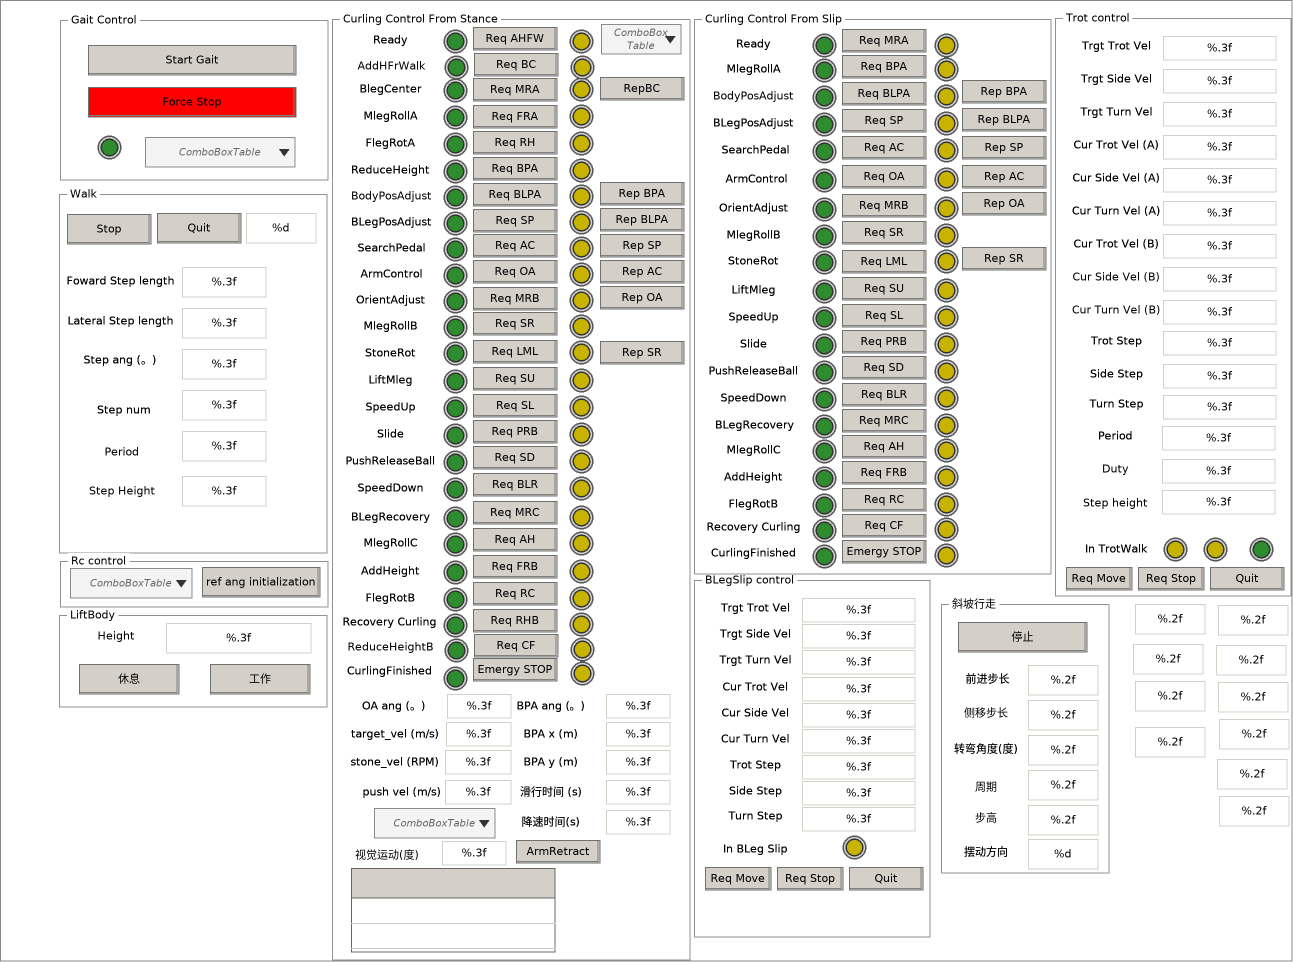
VISUALIZATION RobotUI  // 1293x962
    GroupBox (60,12 268x168), "Gait Control"
        Button (28,33 208x30), "Start Gait", input disabled if: GVL.isInGaitMode
            toggle GVL.startGaitButton
        Button (28,75 208x30), "Force Stop"
            toggle GVL.emergencyStop
        Lamp1 (36,121 27x29), variable: GVL.isInGaitMode, style: Lamp-Lamp1-Green
        ComboBoxTable (85,125 150x30), variable: GVL.gaitId, data array: GVL.gaitNameLists
            p3854506369: GVL.gaitNameLists[INDEX]
    Button (88,45 208x30), "Start Gait", input disabled if: GVL.isInGaitMode
        toggle GVL.startGaitButton
    Button (88,87 208x30), "Force Stop"
        toggle GVL.emergencyStop
    Lamp1 (96,133 27x29), variable: GVL.isInGaitMode, style: Lamp-Lamp1-Green
    ComboBoxTable (145,137 150x30), variable: GVL.gaitId, data array: GVL.gaitNameLists
        p3854506369: GVL.gaitNameLists[INDEX]
    GroupBox (59,186 268x367), "Walk"
        Button (8,28 84x30), "Stop"
            toggle GVL.gaitPlanner.StaticwalkGaitPlanner.require_stop_flag
        Button (98,27 84x30), "Quit"
            toggle GVL.gaitPlanner.StaticwalkGaitPlanner.quit_flag
        Textfield (123,81 84x30), "%.3f", text variable: GVL.gaitPlanner.StaticwalkGaitPlanner.L
            OnMouseClick: write the text variable via Default
        Label (8,80 107x30), "Foward Step length"
        Textfield (123,245 84x30), "%.3f", text variable: GVL.gaitPlanner.StaticwalkGaitPlanner.period
            OnMouseClick: write the text variable via Default
        Textfield (123,290 84x30), "%.3f", text variable: GVL.gaitPlanner.StaticwalkGaitPlanner.H
            OnMouseClick: write the text variable via Default
        Label (21,159 80x30), "Step ang (。)"
        Textfield (123,163 84x30), "%.3f", text variable: GVL.gaitPlanner.StaticwalkGaitPlanner.Yaw
            OnMouseClick: write the text variable via Default
        Label (25,209 80x30), "Step num"
        Textfield (123,204 84x30), "%.3f", text variable: GVL.gaitPlanner.StaticwalkGaitPlanner.N
            OnMouseClick: write the text variable via Default
        Textfield (123,122 84x30), "%.3f", text variable: GVL.gaitPlanner.StaticwalkGaitPlanner.La
            OnMouseClick: write the text variable via Default
        Label (8,120 107x30), "Lateral Step length"
    Button (67,214 84x30), "Stop"
        toggle GVL.gaitPlanner.StaticwalkGaitPlanner.require_stop_flag
    Button (157,213 84x30), "Quit"
        toggle GVL.gaitPlanner.StaticwalkGaitPlanner.quit_flag
    Textfield (182,267 84x30), "%.3f", text variable: GVL.gaitPlanner.StaticwalkGaitPlanner.L
        OnMouseClick: write the text variable via Default
    Label (67,266 107x30), "Foward Step length"
    Textfield (182,431 84x30), "%.3f", text variable: GVL.gaitPlanner.StaticwalkGaitPlanner.period
        OnMouseClick: write the text variable via Default
    Textfield (182,476 84x30), "%.3f", text variable: GVL.gaitPlanner.StaticwalkGaitPlanner.H
        OnMouseClick: write the text variable via Default
    Label (80,345 80x30), "Step ang (。)"
    Textfield (182,349 84x30), "%.3f", text variable: GVL.gaitPlanner.StaticwalkGaitPlanner.Yaw
        OnMouseClick: write the text variable via Default
    Label (84,395 80x30), "Step num"
    Textfield (182,390 84x30), "%.3f", text variable: GVL.gaitPlanner.StaticwalkGaitPlanner.N
        OnMouseClick: write the text variable via Default
    Textfield (182,308 84x30), "%.3f", text variable: GVL.gaitPlanner.StaticwalkGaitPlanner.La
        OnMouseClick: write the text variable via Default
    Label (67,306 107x30), "Lateral Step length"
    GroupBox (59,607 268x100), "LiftBody"
        Label (25,14 64x30), "Height"
        Textfield (107,16 145x30), "%.3f", text variable: GVL.ReduceDistance
            OnMouseClick: write the text variable via Default, min -0.3, max 0.3
        Button (20,57 100x30), "休息"
            toggle gvl.RestButton
        Button (151,57 100x30), "工作"
            toggle gvl.WorkButton
    Label (82,437 80x30), "Period"
    Label (77,476 90x30), "Step Height"
    Textfield (246,213 70x30), "%d", text variable: GVL.gaitPlanner.StaticwalkGaitPlanner.gait_cycle
    GroupBox (332,11 358x949), "Curling Control From Stance"
        Label (4,680 116x30), "OA ang (。)"
        Label (5,14 107x30), "Ready"
        Label (5,63 107x30), "BlegCenter"
        Label (5,90 107x30), "MlegRollA"
        Label (5,117 107x30), "FlegRotA"
        Label (5,144 107x30), "ReduceHeight"
        Label (5,300 107x30), "MlegRollB"
        Label (5,327 107x30), "StoneRot"
        Label (5,354 107x30), "LiftMleg"
        Label (5,381 107x30), "SpeedUp"
        Label (5,408 107x30), "Slide"
        Label (5,435 107x30), "PushReleaseBall"
        Label (5,462 107x30), "SpeedDown"
        Label (5,545 107x30), "AddHeight"
        Label (5,517 107x30), "MlegRollC"
        Label (5,572 107x30), "FlegRotB"
        Label (4,645 107x30), "CurlingFinished"
        Lamp1 (110,16 27x29), variable: GVL.gaitPlanner.CurlingGaitPlanner2.IsReady, style: Lamp-Lamp1-Green
        Lamp1 (110,65 27x29), variable: GVL.gaitPlanner.CurlingGaitPlanner2.IsBlegCenter, style: Lamp-Lamp1-Green
        Lamp1 (110,92 27x29), variable: GVL.gaitPlanner.CurlingGaitPlanner2.IsMlegRollA, style: Lamp-Lamp1-Green
        Lamp1 (110,119 27x29), variable: GVL.gaitPlanner.CurlingGaitPlanner2.IsFlegRotA, style: Lamp-Lamp1-Green
        Lamp1 (110,146 27x29), variable: GVL.gaitPlanner.CurlingGaitPlanner2.IsReduceHeight, style: Lamp-Lamp1-Green
        Lamp1 (110,302 27x29), variable: GVL.gaitPlanner.CurlingGaitPlanner2.IsMlegRollB, style: Lamp-Lamp1-Green
        Lamp1 (110,328 27x29), variable: GVL.gaitPlanner.CurlingGaitPlanner2.IsStoneRot, style: Lamp-Lamp1-Green
        Lamp1 (110,356 27x29), variable: GVL.gaitPlanner.CurlingGaitPlanner2.IsLiftMleg, style: Lamp-Lamp1-Green
        Lamp1 (110,383 27x29), variable: GVL.gaitPlanner.CurlingGaitPlanner2.IsSpeedUp, style: Lamp-Lamp1-Green
        Lamp1 (110,410 27x29), variable: GVL.gaitPlanner.CurlingGaitPlanner2.IsSlide, style: Lamp-Lamp1-Green
        Lamp1 (110,437 27x29), variable: GVL.gaitPlanner.CurlingGaitPlanner2.IsPushReleaseBall, style: Lamp-Lamp1-Green
        Lamp1 (110,464 27x29), variable: GVL.gaitPlanner.CurlingGaitPlanner2.IsSpeedDown, style: Lamp-Lamp1-Green
        Lamp1 (110,519 27x29), variable: GVL.gaitPlanner.CurlingGaitPlanner2.IsMlegRollC, style: Lamp-Lamp1-Green
        Lamp1 (110,547 27x29), variable: GVL.gaitPlanner.CurlingGaitPlanner2.IsAddHeight, style: Lamp-Lamp1-Green
        Lamp1 (110,574 27x29), variable: GVL.gaitPlanner.CurlingGaitPlanner2.IsFlegRotB, style: Lamp-Lamp1-Green
        Lamp1 (110,653 27x29), variable: GVL.gaitPlanner.CurlingGaitPlanner2.IsCurlingFinished, style: Lamp-Lamp1-Green
        Button (141,16 84x23), "Req BC"
            toggle GVL.gaitPlanner.CurlingGaitPlanner2.RequireBlegCenter
        Button (141,67 84x23), "Req MRA"
            toggle GVL.gaitPlanner.CurlingGaitPlanner2.RequireMlegRollA
        Button (141,94 84x23), "Req FRA"
            toggle GVL.gaitPlanner.CurlingGaitPlanner2.RequireFlegRotA
        Button (141,120 84x23), "Req RH"
            toggle GVL.gaitPlanner.CurlingGaitPlanner2.RequireReduceHeight
        Button (141,146 84x23), "Req BPA"
            toggle GVL.gaitPlanner.CurlingGaitPlanner2.RequireBodyPosAdjust
        Button (141,301 84x23), "Req SR"
            toggle GVL.gaitPlanner.CurlingGaitPlanner2.RequireStoneRot
        Button (141,329 84x23), "Req LML"
            toggle GVL.gaitPlanner.CurlingGaitPlanner2.RequireLiftMleg
        Button (141,356 84x23), "Req SU"
            toggle GVL.gaitPlanner.CurlingGaitPlanner2.RequireSpeedUp
        Button (141,383 84x23), "Req SL"
            toggle GVL.gaitPlanner.CurlingGaitPlanner2.RequireSlide
        Button (141,409 84x23), "Req PRB"
            toggle GVL.gaitPlanner.CurlingGaitPlanner2.RequirePushReleaseBall
        Button (141,435 84x23), "Req SD"
            toggle GVL.gaitPlanner.CurlingGaitPlanner2.RequireSpeedDown
        Button (141,462 84x23), "Req BLR"
            toggle GVL.gaitPlanner.CurlingGaitPlanner2.RequireBLegRecovery
        Button (141,517 84x23), "Req AH"
            toggle GVL.gaitPlanner.CurlingGaitPlanner2.RequireAddHeight
        Button (141,544 84x23), "Req FRB"
            toggle GVL.gaitPlanner.CurlingGaitPlanner2.RequireFlegRotB
        Button (141,571 84x23), "Req RC"
            toggle GVL.gaitPlanner.CurlingGaitPlanner2.RequireRecovery
        Button (141,647 84x23), "Emergy STOP"
            toggle GVL.gaitPlanner.CurlingGaitPlanner2.quit_flag
        Label (5,708 116x30), "target_vel (m/s)"
        Label (5,736 116x30), "stone_vel (RPM)"
        Textfield (115,683 64x24), "%.3f", text variable: GVL.adjust_angle_degree
            OnMouseClick: write the text variable via Default
        Textfield (114,711 65x24), "%.3f", text variable: GVL.target_vel
            OnMouseClick: write the text variable via Default
        Textfield (113,739 66x24), "%.3f", text variable: GVL.stone_rot_vel
            OnMouseClick: write the text variable via Default
        Lamp1 (236,64 27x29), variable: GVL.gaitPlanner.CurlingGaitPlanner2.BlegCenterFinished, style: Lamp-Lamp1-Yellow
        Lamp1 (236,91 27x29), variable: GVL.gaitPlanner.CurlingGaitPlanner2.MlegRollAFinished, style: Lamp-Lamp1-Yellow
        Lamp1 (236,118 27x29), variable: GVL.gaitPlanner.CurlingGaitPlanner2.FlegRotAFinished, style: Lamp-Lamp1-Yellow
        Lamp1 (236,145 27x29), variable: GVL.gaitPlanner.CurlingGaitPlanner2.ReduceHeightFinished, style: Lamp-Lamp1-Yellow
        Lamp1 (236,301 27x29), variable: GVL.gaitPlanner.CurlingGaitPlanner2.MlegRollBFinished, style: Lamp-Lamp1-Yellow
        Lamp1 (236,327 27x29), variable: GVL.gaitPlanner.CurlingGaitPlanner2.StoneRotFinished, style: Lamp-Lamp1-Yellow
        Lamp1 (236,355 27x29), variable: GVL.gaitPlanner.CurlingGaitPlanner2.LiftMlegFinished, style: Lamp-Lamp1-Yellow
        Lamp1 (236,382 27x29), variable: GVL.gaitPlanner.CurlingGaitPlanner2.SpeedUpFinished, style: Lamp-Lamp1-Yellow
        Lamp1 (236,409 27x29), variable: GVL.gaitPlanner.CurlingGaitPlanner2.SlideFinished, style: Lamp-Lamp1-Yellow
        Lamp1 (236,436 27x29), variable: GVL.gaitPlanner.CurlingGaitPlanner2.PushReleaseBallFinished, style: Lamp-Lamp1-Yellow
        Lamp1 (236,463 27x29), variable: GVL.gaitPlanner.CurlingGaitPlanner2.SpeedDownFinished, style: Lamp-Lamp1-Yellow
        Lamp1 (236,518 27x29), variable: GVL.gaitPlanner.CurlingGaitPlanner2.MlegRollCFinished, style: Lamp-Lamp1-Yellow
        Lamp1 (236,546 27x29), variable: GVL.gaitPlanner.CurlingGaitPlanner2.AddHeightFinished, style: Lamp-Lamp1-Yellow
        Lamp1 (236,573 27x29), variable: GVL.gaitPlanner.CurlingGaitPlanner2.FlegRotBFinished, style: Lamp-Lamp1-Yellow
        Lamp1 (237,648 27x29), variable: GVL.gaitPlanner.CurlingGaitPlanner2.CurlingGaitFinished, style: Lamp-Lamp1-Yellow
        Lamp1 (236,16 27x29), variable: GVL.gaitPlanner.CurlingGaitPlanner2.ReadyFinished, style: Lamp-Lamp1-Yellow
        Label (12,766 116x30), "push vel (m/s)"
        Textfield (113,769 66x24), "%.3f", text variable: gvl.PushVelocityIn
            OnMouseClick: write the text variable via Default
        Button (268,66 84x23), "RepBC"
            toggle GVL.gaitPlanner.CurlingGaitPlanner2.RequireRepeateBlegCenter
        Button (268,330 84x23), "Rep SR"
            toggle GVL.gaitPlanner.CurlingGaitPlanner2.RequireRepeateStoneRot
        Button (268,275 84x23), "Rep OA"
            toggle GVL.gaitPlanner.CurlingGaitPlanner2.RequireRepeateOrientAdjust
        Label (5,274 107x30), "OrientAdjust"
        Label (6,222 107x30), "SearchPedal"
        Button (268,197 84x23), "Rep BLPA"
            toggle GVL.gaitPlanner.CurlingGaitPlanner2.RequireRepeateBLegPosAdjust
        Label (161,680 116x30), "BPA ang (。)"
        Label (161,708 116x30), "BPA x (m)"
        Label (161,736 116x30), "BPA y (m)"
        Textfield (274,683 64x24), "%.3f", text variable: GVL.BPA_adjust_angle_degree
            OnMouseClick: write the text variable via Default
        Textfield (274,711 64x24), "%.3f", text variable: GVL.BPA_adjust_x
            OnMouseClick: write the text variable via Default
        Textfield (274,739 64x24), "%.3f", text variable: GVL.BPA_adjust_y
            OnMouseClick: write the text variable via Default
        Button (740,-63 84x23), "RepBC"
            toggle GVL.gaitPlanner.CurlingGaitPlanner2.RequireRepeateBlegCenter
        ComboBoxTable (42,797 121x30), variable: gvl.curlingPushModel, data array: gvl.curlingPushModelList
            p3854506369: gvl.curlingPushModelList[INDEX]
        Label (161,766 116x30), "滑行时间 (s)"
        Label (161,796 116x30), "降速时间(s)"
        Textfield (274,769 64x24), "%.3f", text variable: GVL.slideTimeIn
            OnMouseClick: write the text variable via Default
        Textfield (274,799 64x24), "%.3f", text variable: GVL.PushFinishDurationTimeIn
            OnMouseClick: write the text variable via Default
        Label (4,596 107x30), "Recovery Curling"
        Label (6,196 107x30), "BLegPosAdjust"
        Button (268,223 84x23), "Rep SP"
            toggle GVL.gaitPlanner.CurlingGaitPlanner2.RequireRepeateSearchPedal
        Button (184,829 84x23), "ArmRetract"
            toggle GVL.ArmRetractControl
        Label (6,248 107x30), "ArmControl"
        Textfield (110,830 64x24), "%.3f", text variable: GVL.AC_AngleDegIn
            OnMouseClick: write the text variable via Default
        Button (268,249 84x23), "Rep AC"
            toggle GVL.gaitPlanner.CurlingGaitPlanner2.RequireRepeateArmControl
        Label (5,491 107x30), "BLegRecovery"
        Label (370,124 107x30), "SearchPedal"
        Label (371,153 107x30), "ArmControl"
        Label (369,399 107x30), "BLegRecovery"
        Label (368,501 107x30), "Recovery Curling"
        Table (19,857 204x84), data array: GVL.BLPA_adjust_distance_desire
            p3854506369: GVL.BLPA_adjust_distance_desire[0,INDEX]
            p1892666644: GVL.BLPA_adjust_distance_desire[1,INDEX]
            p2232123230: LegA AdjInc
            p511219082: LegF AdjInc
            Columns.Column.[0].Template: OnMouseClick: write the text variable via Default
            Columns.Column.[1].Template: OnMouseClick: write the text variable via Default
        Label (5,621 107x30), "ReduceHeightB"
        Label (6,40 107x30), "AddHFrWalk"
        ComboBoxTable (269,13 80x30), variable: GVL.taskChooseId, data array: gvl.taskChooseList
            p3854506369: gvl.taskChooseList[INDEX]
    Label (336,691 116x30), "OA ang (。)"
    Label (337,25 107x30), "Ready"
    Label (337,74 107x30), "BlegCenter"
    Label (337,101 107x30), "MlegRollA"
    Label (337,128 107x30), "FlegRotA"
    Label (337,155 107x30), "ReduceHeight"
    Label (337,311 107x30), "MlegRollB"
    Label (337,338 107x30), "StoneRot"
    Label (337,365 107x30), "LiftMleg"
    Label (337,392 107x30), "SpeedUp"
    Label (337,419 107x30), "Slide"
    Label (337,446 107x30), "PushReleaseBall"
    Label (337,473 107x30), "SpeedDown"
    Label (337,556 107x30), "AddHeight"
    Label (337,528 107x30), "MlegRollC"
    Label (337,583 107x30), "FlegRotB"
    Label (336,656 107x30), "CurlingFinished"
    Lamp1 (442,27 27x29), variable: GVL.gaitPlanner.CurlingGaitPlanner2.IsReady, style: Lamp-Lamp1-Green
    Lamp1 (442,76 27x29), variable: GVL.gaitPlanner.CurlingGaitPlanner2.IsBlegCenter, style: Lamp-Lamp1-Green
    Lamp1 (442,103 27x29), variable: GVL.gaitPlanner.CurlingGaitPlanner2.IsMlegRollA, style: Lamp-Lamp1-Green
    Lamp1 (442,130 27x29), variable: GVL.gaitPlanner.CurlingGaitPlanner2.IsFlegRotA, style: Lamp-Lamp1-Green
    Lamp1 (442,157 27x29), variable: GVL.gaitPlanner.CurlingGaitPlanner2.IsReduceHeight, style: Lamp-Lamp1-Green
    Lamp1 (442,313 27x29), variable: GVL.gaitPlanner.CurlingGaitPlanner2.IsMlegRollB, style: Lamp-Lamp1-Green
    Lamp1 (442,339 27x29), variable: GVL.gaitPlanner.CurlingGaitPlanner2.IsStoneRot, style: Lamp-Lamp1-Green
    Lamp1 (442,367 27x29), variable: GVL.gaitPlanner.CurlingGaitPlanner2.IsLiftMleg, style: Lamp-Lamp1-Green
    Lamp1 (442,394 27x29), variable: GVL.gaitPlanner.CurlingGaitPlanner2.IsSpeedUp, style: Lamp-Lamp1-Green
    Lamp1 (442,421 27x29), variable: GVL.gaitPlanner.CurlingGaitPlanner2.IsSlide, style: Lamp-Lamp1-Green
    Lamp1 (442,448 27x29), variable: GVL.gaitPlanner.CurlingGaitPlanner2.IsPushReleaseBall, style: Lamp-Lamp1-Green
    Lamp1 (442,475 27x29), variable: GVL.gaitPlanner.CurlingGaitPlanner2.IsSpeedDown, style: Lamp-Lamp1-Green
    Lamp1 (442,530 27x29), variable: GVL.gaitPlanner.CurlingGaitPlanner2.IsMlegRollC, style: Lamp-Lamp1-Green
    Lamp1 (442,558 27x29), variable: GVL.gaitPlanner.CurlingGaitPlanner2.IsAddHeight, style: Lamp-Lamp1-Green
    Lamp1 (442,585 27x29), variable: GVL.gaitPlanner.CurlingGaitPlanner2.IsFlegRotB, style: Lamp-Lamp1-Green
    Lamp1 (442,664 27x29), variable: GVL.gaitPlanner.CurlingGaitPlanner2.IsCurlingFinished, style: Lamp-Lamp1-Green
    Button (473,27 84x23), "Req AHFW"
        toggle GVL.gaitPlanner.CurlingGaitPlanner2.RequireAddHeightFromWalk
    Button (473,78 84x23), "Req MRA"
        toggle GVL.gaitPlanner.CurlingGaitPlanner2.RequireMlegRollA
    Button (473,105 84x23), "Req FRA"
        toggle GVL.gaitPlanner.CurlingGaitPlanner2.RequireFlegRotA
    Button (473,131 84x23), "Req RH"
        toggle GVL.gaitPlanner.CurlingGaitPlanner2.RequireReduceHeight
    Button (473,157 84x23), "Req BPA"
        toggle GVL.gaitPlanner.CurlingGaitPlanner2.RequireBodyPosAdjust
    Button (473,312 84x23), "Req SR"
        toggle GVL.gaitPlanner.CurlingGaitPlanner2.RequireStoneRot
    Button (473,340 84x23), "Req LML"
        toggle GVL.gaitPlanner.CurlingGaitPlanner2.RequireLiftMleg
    Button (473,367 84x23), "Req SU"
        toggle GVL.gaitPlanner.CurlingGaitPlanner2.RequireSpeedUp
    Button (473,394 84x23), "Req SL"
        toggle GVL.gaitPlanner.CurlingGaitPlanner2.RequireSlide
    Button (473,420 84x23), "Req PRB"
        toggle GVL.gaitPlanner.CurlingGaitPlanner2.RequirePushReleaseBall
    Button (473,446 84x23), "Req SD"
        toggle GVL.gaitPlanner.CurlingGaitPlanner2.RequireSpeedDown
    Button (473,473 84x23), "Req BLR"
        toggle GVL.gaitPlanner.CurlingGaitPlanner2.RequireBLegRecovery
    Button (473,528 84x23), "Req AH"
        toggle GVL.gaitPlanner.CurlingGaitPlanner2.RequireAddHeight
    Button (473,555 84x23), "Req FRB"
        toggle GVL.gaitPlanner.CurlingGaitPlanner2.RequireFlegRotB
    Button (473,582 84x23), "Req RC"
        toggle GVL.gaitPlanner.CurlingGaitPlanner2.RequireRecovery
    Button (473,658 84x23), "Emergy STOP"
        toggle GVL.gaitPlanner.CurlingGaitPlanner2.quit_flag
    Label (337,719 116x30), "target_vel (m/s)"
    Label (337,747 116x30), "stone_vel (RPM)"
    Textfield (447,694 64x24), "%.3f", text variable: GVL.adjust_angle_degree
        OnMouseClick: write the text variable via Default, min -6, max 6
    Textfield (446,722 65x24), "%.3f", text variable: GVL.target_vel
        OnMouseClick: write the text variable via Default, min 0.5, max 2.5
    Textfield (445,750 66x24), "%.3f", text variable: GVL.stone_rot_vel
        OnMouseClick: write the text variable via Default, min -80, max 80
    Lamp1 (568,75 27x29), variable: GVL.gaitPlanner.CurlingGaitPlanner2.BlegCenterFinished, style: Lamp-Lamp1-Yellow
    Lamp1 (568,102 27x29), variable: GVL.gaitPlanner.CurlingGaitPlanner2.MlegRollAFinished, style: Lamp-Lamp1-Yellow
    Lamp1 (568,129 27x29), variable: GVL.gaitPlanner.CurlingGaitPlanner2.FlegRotAFinished, style: Lamp-Lamp1-Yellow
    Lamp1 (568,156 27x29), variable: GVL.gaitPlanner.CurlingGaitPlanner2.ReduceHeightFinished, style: Lamp-Lamp1-Yellow
    Lamp1 (568,312 27x29), variable: GVL.gaitPlanner.CurlingGaitPlanner2.MlegRollBFinished, style: Lamp-Lamp1-Yellow
    Lamp1 (568,338 27x29), variable: GVL.gaitPlanner.CurlingGaitPlanner2.StoneRotFinished, style: Lamp-Lamp1-Yellow
    Lamp1 (568,366 27x29), variable: GVL.gaitPlanner.CurlingGaitPlanner2.LiftMlegFinished, style: Lamp-Lamp1-Yellow
    Lamp1 (568,393 27x29), variable: GVL.gaitPlanner.CurlingGaitPlanner2.SpeedUpFinished, style: Lamp-Lamp1-Yellow
    Lamp1 (568,420 27x29), variable: GVL.gaitPlanner.CurlingGaitPlanner2.SlideFinished, style: Lamp-Lamp1-Yellow
    Lamp1 (568,447 27x29), variable: GVL.gaitPlanner.CurlingGaitPlanner2.PushReleaseBallFinished, style: Lamp-Lamp1-Yellow
    Lamp1 (568,474 27x29), variable: GVL.gaitPlanner.CurlingGaitPlanner2.SpeedDownFinished, style: Lamp-Lamp1-Yellow
    Lamp1 (568,529 27x29), variable: GVL.gaitPlanner.CurlingGaitPlanner2.MlegRollCFinished, style: Lamp-Lamp1-Yellow
    Lamp1 (568,557 27x29), variable: GVL.gaitPlanner.CurlingGaitPlanner2.AddHeightFinished, style: Lamp-Lamp1-Yellow
    Lamp1 (568,584 27x29), variable: GVL.gaitPlanner.CurlingGaitPlanner2.FlegRotBFinished, style: Lamp-Lamp1-Yellow
    Lamp1 (569,659 27x29), variable: GVL.gaitPlanner.CurlingGaitPlanner2.CurlingGaitFinished, style: Lamp-Lamp1-Yellow
    Lamp1 (568,27 27x29), variable: GVL.gaitPlanner.CurlingGaitPlanner2.ReadyFinished, style: Lamp-Lamp1-Yellow
    Label (344,777 116x30), "push vel (m/s)"
    Textfield (445,780 66x24), "%.3f", text variable: gvl.PushVelocityIn
        OnMouseClick: write the text variable via Default, min 0.5, max 2.7
    Button (600,77 84x23), "RepBC"
        toggle GVL.gaitPlanner.CurlingGaitPlanner2.RequireRepeateBlegCenter
    Button (600,341 84x23), "Rep SR"
        toggle GVL.gaitPlanner.CurlingGaitPlanner2.RequireRepeateStoneRot
    Button (600,286 84x23), "Rep OA"
        toggle GVL.gaitPlanner.CurlingGaitPlanner2.RequireRepeateOrientAdjust
    Label (337,285 107x30), "OrientAdjust"
    Label (338,233 107x30), "SearchPedal"
    Button (600,208 84x23), "Rep BLPA"
        toggle GVL.gaitPlanner.CurlingGaitPlanner2.RequireRepeateBLegPosAdjust
    Label (493,691 116x30), "BPA ang (。)"
    Label (493,719 116x30), "BPA x (m)"
    Label (493,747 116x30), "BPA y (m)"
    Textfield (606,694 64x24), "%.3f", text variable: GVL.BPA_adjust_angle_degree
        OnMouseClick: write the text variable via Default, min -6, max 6
    Textfield (606,722 64x24), "%.3f", text variable: GVL.BPA_adjust_x
        OnMouseClick: write the text variable via Default, min -0.1, max 0.1
    Textfield (606,750 64x24), "%.3f", text variable: GVL.BPA_adjust_y
        OnMouseClick: write the text variable via Default, min -0.05, max 0.05
    ComboBoxTable (374,808 121x30), variable: gvl.curlingPushModel, data array: gvl.curlingPushModelList
        p3854506369: gvl.curlingPushModelList[INDEX]
    Label (493,777 116x30), "滑行时间 (s)"
    Label (493,807 116x30), "降速时间(s)"
    Textfield (606,780 64x24), "%.3f", text variable: GVL.slideTimeIn
        OnMouseClick: write the text variable via Default, min 0.1, max 5
    Textfield (606,810 64x24), "%.3f", text variable: GVL.PushFinishDurationTimeIn
        OnMouseClick: write the text variable via Default, min 0.1, max 10
    Label (336,607 107x30), "Recovery Curling"
    Label (338,207 107x30), "BLegPosAdjust"
    Button (600,234 84x23), "Rep SP"
        toggle GVL.gaitPlanner.CurlingGaitPlanner2.RequireRepeateSearchPedal
    Button (516,840 84x23), "ArmRetract"
        toggle GVL.ArmRetractControl
    Label (338,259 107x30), "ArmControl"
    Textfield (442,841 64x24), "%.3f", text variable: GVL.AC_AngleDegIn
        OnMouseClick: write the text variable via Default, min -60, max 0
    Button (600,260 84x23), "Rep AC"
        toggle GVL.gaitPlanner.CurlingGaitPlanner2.RequireRepeateArmControl
    Label (337,502 107x30), "BLegRecovery"
    Label (702,135 107x30), "SearchPedal"
    Label (703,164 107x30), "ArmControl"
    Label (701,410 107x30), "BLegRecovery"
    Label (700,512 107x30), "Recovery Curling"
    Table (351,868 204x84), data array: GVL.BLPA_adjust_distance_desire
        p3854506369: GVL.BLPA_adjust_distance_desire[0,INDEX]
        p1892666644: GVL.BLPA_adjust_distance_desire[1,INDEX]
        p2232123230: LegA AdjInc
        p511219082: LegF AdjInc
        Columns.Column.[0].Template: OnMouseClick: write the text variable via Default
        Columns.Column.[1].Template: OnMouseClick: write the text variable via Default
    GroupBox (60,553 268x54), "Rc control"
        Button (142,14 118x30), "ref ang initialization"
            toggle gvl.setRcRefAngButton
        ComboBoxTable (10,15 122x30), variable: gvl.RcGaitId, data array: GVL.RcGaitNameLists
            p3854506369: GVL.RcGaitNameLists[INDEX]
    Button (202,567 118x30), "ref ang initialization"
        toggle gvl.setRcRefAngButton
    ComboBoxTable (70,568 122x30), variable: gvl.RcGaitId, data array: GVL.RcGaitNameLists
        p3854506369: GVL.RcGaitNameLists[INDEX]
    GroupBox (694,572 236x365), "BLegSlip control"
        Label (8,21 107x30), "Trgt Trot Vel"
        Label (8,47 107x30), "Trgt Side Vel"
        Label (8,73 107x30), "Trgt Turn Vel"
        Textfield (108,26 113x24), "%.3f", text variable: GVL.BLegSlip_trot_vel_desire
            OnMouseClick: write the text variable via Default
        Textfield (108,52 113x24), "%.3f", text variable: GVL.BLegSlip_side_vel_desire
            OnMouseClick: write the text variable via Default
        Textfield (108,78 113x24), "%.3f", text variable: GVL.BLegSlip_turn_rate_desire
            OnMouseClick: write the text variable via Default
        Label (8,100 107x30), "Cur Trot Vel"
        Label (8,126 107x30), "Cur Side Vel"
        Label (8,152 107x30), "Cur Turn Vel"
        Textfield (108,105 113x24), "%.3f", text variable: GVL.gaitPlanner.BLegSlipPlanner.trot_vel
        Textfield (108,131 113x24), "%.3f", text variable: GVL.gaitPlanner.BLegSlipPlanner.side_vel
        Textfield (108,157 113x24), "%.3f", text variable: GVL.gaitPlanner.BLegSlipPlanner.turn_rate
        Label (8,178 107x30), "Trot Step"
        Label (8,204 107x30), "Side Step"
        Label (8,229 107x30), "Turn Step"
        Textfield (108,183 113x24), "%.3f", text variable: GVL.BLegSlip_step[0]
            OnMouseClick: write the text variable via Default
        Textfield (108,209 113x24), "%.3f", text variable: GVL.BLegSlip_step[1]
            OnMouseClick: write the text variable via Default
        Textfield (108,235 113x24), "%.3f", text variable: GVL.BLegSlip_step[2]
            OnMouseClick: write the text variable via Default
        Button (11,295 66x23), "Req Move"
            toggle GVL.gaitPlanner.BLegSlipPlanner.require_move
        Button (83,295 66x23), "Req Stop"
            toggle GVL.gaitPlanner.BLegSlipPlanner.requir_stop
        Button (155,295 74x23), "Quit"
            toggle GVL.gaitPlanner.BLegSlipPlanner.quit_flag
        Label (8,262 107x30), "In BLeg Slip"
        Lamp1 (147,261 27x29), variable: GVL.gaitPlanner.BLegSlipPlanner.inSlip, style: Lamp-Lamp1-Yellow
    Label (702,593 107x30), "Trgt Trot Vel"
    Label (702,619 107x30), "Trgt Side Vel"
    Label (702,645 107x30), "Trgt Turn Vel"
    Textfield (802,598 113x24), "%.3f", text variable: GVL.BLegSlip_trot_vel_desire
        OnMouseClick: write the text variable via Default
    Textfield (802,624 113x24), "%.3f", text variable: GVL.BLegSlip_side_vel_desire
        OnMouseClick: write the text variable via Default
    Textfield (802,650 113x24), "%.3f", text variable: GVL.BLegSlip_turn_rate_desire
        OnMouseClick: write the text variable via Default
    Label (702,672 107x30), "Cur Trot Vel"
    Label (702,698 107x30), "Cur Side Vel"
    Label (702,724 107x30), "Cur Turn Vel"
    Textfield (802,677 113x24), "%.3f", text variable: GVL.gaitPlanner.BLegSlipPlanner.trot_vel
    Textfield (802,703 113x24), "%.3f", text variable: GVL.gaitPlanner.BLegSlipPlanner.side_vel
    Textfield (802,729 113x24), "%.3f", text variable: GVL.gaitPlanner.BLegSlipPlanner.turn_rate
    Label (702,750 107x30), "Trot Step"
    Label (702,776 107x30), "Side Step"
    Label (702,801 107x30), "Turn Step"
    Textfield (802,755 113x24), "%.3f", text variable: GVL.BLegSlip_step[0]
        OnMouseClick: write the text variable via Default
    Textfield (802,781 113x24), "%.3f", text variable: GVL.BLegSlip_step[1]
        OnMouseClick: write the text variable via Default
    Textfield (802,807 113x24), "%.3f", text variable: GVL.BLegSlip_step[2]
        OnMouseClick: write the text variable via Default
    Button (705,867 66x23), "Req Move"
        toggle GVL.gaitPlanner.BLegSlipPlanner.require_move
    Button (777,867 66x23), "Req Stop"
        toggle GVL.gaitPlanner.BLegSlipPlanner.requir_stop
    Button (849,867 74x23), "Quit"
        toggle GVL.gaitPlanner.BLegSlipPlanner.quit_flag
    Label (702,834 107x30), "In BLeg Slip"
    Lamp1 (841,833 27x29), variable: GVL.gaitPlanner.BLegSlipPlanner.inSlip, style: Lamp-Lamp1-Yellow
    GroupBox (694,11 357x563), "Curling Control From Slip"
        Label (6,18 107x30), "Ready"
        Label (6,43 107x30), "MlegRollA"
        Label (6,235 107x30), "StoneRot"
        Label (6,264 107x30), "LiftMleg"
        Label (6,291 107x30), "SpeedUp"
        Label (6,318 107x30), "Slide"
        Label (6,345 107x30), "PushReleaseBall"
        Label (6,372 107x30), "SpeedDown"
        Label (6,451 107x30), "AddHeight"
        Label (6,424 107x30), "MlegRollC"
        Label (6,478 107x30), "FlegRotB"
        Label (6,527 107x30), "CurlingFinished"
        Lamp1 (117,20 27x29), variable: GVL.gaitPlanner.CurlingGaitFromSlipPlanner.IsReady, style: Lamp-Lamp1-Green
        Lamp1 (117,45 27x29), variable: GVL.gaitPlanner.CurlingGaitFromSlipPlanner.IsMlegRollA, style: Lamp-Lamp1-Green
        Lamp1 (117,237 27x29), variable: GVL.gaitPlanner.CurlingGaitFromSlipPlanner.IsStoneRot, style: Lamp-Lamp1-Green
        Lamp1 (117,266 27x29), variable: GVL.gaitPlanner.CurlingGaitFromSlipPlanner.IsLiftMleg, style: Lamp-Lamp1-Green
        Lamp1 (117,293 27x29), variable: GVL.gaitPlanner.CurlingGaitFromSlipPlanner.IsSpeedUp, style: Lamp-Lamp1-Green
        Lamp1 (117,320 27x29), variable: GVL.gaitPlanner.CurlingGaitFromSlipPlanner.IsSlide, style: Lamp-Lamp1-Green
        Lamp1 (117,347 27x29), variable: GVL.gaitPlanner.CurlingGaitFromSlipPlanner.IsPushReleaseBall, style: Lamp-Lamp1-Green
        Lamp1 (117,374 27x29), variable: GVL.gaitPlanner.CurlingGaitFromSlipPlanner.IsSpeedDown, style: Lamp-Lamp1-Green
        Lamp1 (117,426 27x29), variable: GVL.gaitPlanner.CurlingGaitFromSlipPlanner.IsMlegRollC, style: Lamp-Lamp1-Green
        Lamp1 (117,453 27x29), variable: GVL.gaitPlanner.CurlingGaitFromSlipPlanner.IsAddHeight, style: Lamp-Lamp1-Green
        Lamp1 (117,480 27x29), variable: GVL.gaitPlanner.CurlingGaitFromSlipPlanner.IsFlegRotB, style: Lamp-Lamp1-Green
        Lamp1 (117,531 27x29), variable: GVL.gaitPlanner.CurlingGaitFromSlipPlanner.IsCurlingFinished, style: Lamp-Lamp1-Green
        Button (148,18 84x23), "Req MRA"
            toggle GVL.gaitPlanner.CurlingGaitFromSlipPlanner.RequireMlegRollA
        Button (148,44 84x23), "Req BPA"
            toggle GVL.gaitPlanner.CurlingGaitFromSlipPlanner.RequireBodyPosAdjust
        Button (148,239 84x23), "Req LML"
            toggle GVL.gaitPlanner.CurlingGaitFromSlipPlanner.RequireLiftMleg
        Button (148,266 84x23), "Req SU"
            toggle GVL.gaitPlanner.CurlingGaitFromSlipPlanner.RequireSpeedUp
        Button (148,293 84x23), "Req SL"
            toggle GVL.gaitPlanner.CurlingGaitFromSlipPlanner.RequireSlide
        Button (148,319 84x23), "Req PRB"
            toggle GVL.gaitPlanner.CurlingGaitFromSlipPlanner.RequirePushReleaseBall
        Button (148,345 84x23), "Req SD"
            toggle GVL.gaitPlanner.CurlingGaitFromSlipPlanner.RequireSpeedDown
        Button (148,372 84x23), "Req BLR"
            toggle GVL.gaitPlanner.CurlingGaitFromSlipPlanner.RequireBLegRecovery
        Button (148,424 84x23), "Req AH"
            toggle GVL.gaitPlanner.CurlingGaitFromSlipPlanner.RequireAddHeight
        Button (148,450 84x23), "Req FRB"
            toggle GVL.gaitPlanner.CurlingGaitFromSlipPlanner.RequireFlegRotB
        Button (148,477 84x23), "Req RC"
            toggle GVL.gaitPlanner.CurlingGaitFromSlipPlanner.RequireRecovery
        Button (148,529 84x23), "Emergy STOP"
            toggle GVL.gaitPlanner.CurlingGaitFromSlipPlanner.quit_flag
        Lamp1 (239,44 27x29), variable: GVL.gaitPlanner.CurlingGaitFromSlipPlanner.MlegRollAFinished, style: Lamp-Lamp1-Yellow
        Lamp1 (239,236 27x29), variable: GVL.gaitPlanner.CurlingGaitFromSlipPlanner.StoneRotFinished, style: Lamp-Lamp1-Yellow
        Lamp1 (239,265 27x29), variable: GVL.gaitPlanner.CurlingGaitFromSlipPlanner.LiftMlegFinished, style: Lamp-Lamp1-Yellow
        Lamp1 (239,292 27x29), variable: GVL.gaitPlanner.CurlingGaitFromSlipPlanner.SpeedUpFinished, style: Lamp-Lamp1-Yellow
        Lamp1 (239,319 27x29), variable: GVL.gaitPlanner.CurlingGaitFromSlipPlanner.SlideFinished, style: Lamp-Lamp1-Yellow
        Lamp1 (239,346 27x29), variable: GVL.gaitPlanner.CurlingGaitFromSlipPlanner.PushReleaseBallFinished, style: Lamp-Lamp1-Yellow
        Lamp1 (239,373 27x29), variable: GVL.gaitPlanner.CurlingGaitFromSlipPlanner.SpeedDownFinished, style: Lamp-Lamp1-Yellow
        Lamp1 (239,425 27x29), variable: GVL.gaitPlanner.CurlingGaitFromSlipPlanner.MlegRollCFinished, style: Lamp-Lamp1-Yellow
        Lamp1 (239,452 27x29), variable: GVL.gaitPlanner.CurlingGaitFromSlipPlanner.AddHeightFinished, style: Lamp-Lamp1-Yellow
        Lamp1 (239,479 27x29), variable: GVL.gaitPlanner.CurlingGaitFromSlipPlanner.FlegRotBFinished, style: Lamp-Lamp1-Yellow
        Lamp1 (239,530 27x29), variable: GVL.gaitPlanner.CurlingGaitFromSlipPlanner.CurlingGaitFinished, style: Lamp-Lamp1-Yellow
        Lamp1 (239,20 27x29), variable: GVL.gaitPlanner.CurlingGaitFromSlipPlanner.ReadyFinished, style: Lamp-Lamp1-Yellow
        Label (6,209 107x30), "MlegRollB"
        Label (6,182 107x30), "OrientAdjust"
        Label (6,97 107x30), "BLegPosAdjust"
        Button (268,236 84x23), "Rep SR"
            toggle GVL.gaitPlanner.CurlingGaitFromSlipPlanner.RequireRepeateStoneRot
        Button (268,181 84x23), "Rep OA"
            toggle GVL.gaitPlanner.CurlingGaitFromSlipPlanner.RequireRepeateOrientAdjust
        Button (268,97 84x23), "Rep BLPA"
            toggle GVL.gaitPlanner.CurlingGaitFromSlipPlanner.RequireRepeateBLegPosAdjust
        Button (268,69 84x23), "Rep BPA"
            toggle GVL.gaitPlanner.CurlingGaitFromSlipPlanner.RequireRepeateBodyPosAdjust
    Label (700,29 107x30), "Ready"
    Label (700,54 107x30), "MlegRollA"
    Label (700,246 107x30), "StoneRot"
    Label (700,275 107x30), "LiftMleg"
    Label (700,302 107x30), "SpeedUp"
    Label (700,329 107x30), "Slide"
    Label (700,356 107x30), "PushReleaseBall"
    Label (700,383 107x30), "SpeedDown"
    Label (700,462 107x30), "AddHeight"
    Label (700,435 107x30), "MlegRollC"
    Label (700,489 107x30), "FlegRotB"
    Label (700,538 107x30), "CurlingFinished"
    Lamp1 (811,31 27x29), variable: GVL.gaitPlanner.CurlingGaitFromSlipPlanner.IsReady, style: Lamp-Lamp1-Green
    Lamp1 (811,56 27x29), variable: GVL.gaitPlanner.CurlingGaitFromSlipPlanner.IsMlegRollA, style: Lamp-Lamp1-Green
    Lamp1 (811,248 27x29), variable: GVL.gaitPlanner.CurlingGaitFromSlipPlanner.IsStoneRot, style: Lamp-Lamp1-Green
    Lamp1 (811,277 27x29), variable: GVL.gaitPlanner.CurlingGaitFromSlipPlanner.IsLiftMleg, style: Lamp-Lamp1-Green
    Lamp1 (811,304 27x29), variable: GVL.gaitPlanner.CurlingGaitFromSlipPlanner.IsSpeedUp, style: Lamp-Lamp1-Green
    Lamp1 (811,331 27x29), variable: GVL.gaitPlanner.CurlingGaitFromSlipPlanner.IsSlide, style: Lamp-Lamp1-Green
    Lamp1 (811,358 27x29), variable: GVL.gaitPlanner.CurlingGaitFromSlipPlanner.IsPushReleaseBall, style: Lamp-Lamp1-Green
    Lamp1 (811,385 27x29), variable: GVL.gaitPlanner.CurlingGaitFromSlipPlanner.IsSpeedDown, style: Lamp-Lamp1-Green
    Lamp1 (811,437 27x29), variable: GVL.gaitPlanner.CurlingGaitFromSlipPlanner.IsMlegRollC, style: Lamp-Lamp1-Green
    Lamp1 (811,464 27x29), variable: GVL.gaitPlanner.CurlingGaitFromSlipPlanner.IsAddHeight, style: Lamp-Lamp1-Green
    Lamp1 (811,491 27x29), variable: GVL.gaitPlanner.CurlingGaitFromSlipPlanner.IsFlegRotB, style: Lamp-Lamp1-Green
    Lamp1 (811,542 27x29), variable: GVL.gaitPlanner.CurlingGaitFromSlipPlanner.IsCurlingFinished, style: Lamp-Lamp1-Green
    Button (842,29 84x23), "Req MRA"
        toggle GVL.gaitPlanner.CurlingGaitFromSlipPlanner.RequireMlegRollA
    Button (842,55 84x23), "Req BPA"
        toggle GVL.gaitPlanner.CurlingGaitFromSlipPlanner.RequireBodyPosAdjust
    Button (842,250 84x23), "Req LML"
        toggle GVL.gaitPlanner.CurlingGaitFromSlipPlanner.RequireLiftMleg
    Button (842,277 84x23), "Req SU"
        toggle GVL.gaitPlanner.CurlingGaitFromSlipPlanner.RequireSpeedUp
    Button (842,304 84x23), "Req SL"
        toggle GVL.gaitPlanner.CurlingGaitFromSlipPlanner.RequireSlide
    Button (842,330 84x23), "Req PRB"
        toggle GVL.gaitPlanner.CurlingGaitFromSlipPlanner.RequirePushReleaseBall
    Button (842,356 84x23), "Req SD"
        toggle GVL.gaitPlanner.CurlingGaitFromSlipPlanner.RequireSpeedDown
    Button (842,383 84x23), "Req BLR"
        toggle GVL.gaitPlanner.CurlingGaitFromSlipPlanner.RequireBLegRecovery
    Button (842,435 84x23), "Req AH"
        toggle GVL.gaitPlanner.CurlingGaitFromSlipPlanner.RequireAddHeight
    Button (842,461 84x23), "Req FRB"
        toggle GVL.gaitPlanner.CurlingGaitFromSlipPlanner.RequireFlegRotB
    Button (842,488 84x23), "Req RC"
        toggle GVL.gaitPlanner.CurlingGaitFromSlipPlanner.RequireRecovery
    Button (842,540 84x23), "Emergy STOP"
        toggle GVL.gaitPlanner.CurlingGaitFromSlipPlanner.quit_flag
    Lamp1 (933,55 27x29), variable: GVL.gaitPlanner.CurlingGaitFromSlipPlanner.MlegRollAFinished, style: Lamp-Lamp1-Yellow
    Lamp1 (933,247 27x29), variable: GVL.gaitPlanner.CurlingGaitFromSlipPlanner.StoneRotFinished, style: Lamp-Lamp1-Yellow
    Lamp1 (933,276 27x29), variable: GVL.gaitPlanner.CurlingGaitFromSlipPlanner.LiftMlegFinished, style: Lamp-Lamp1-Yellow
    Lamp1 (933,303 27x29), variable: GVL.gaitPlanner.CurlingGaitFromSlipPlanner.SpeedUpFinished, style: Lamp-Lamp1-Yellow
    Lamp1 (933,330 27x29), variable: GVL.gaitPlanner.CurlingGaitFromSlipPlanner.SlideFinished, style: Lamp-Lamp1-Yellow
    Lamp1 (933,357 27x29), variable: GVL.gaitPlanner.CurlingGaitFromSlipPlanner.PushReleaseBallFinished, style: Lamp-Lamp1-Yellow
    Lamp1 (933,384 27x29), variable: GVL.gaitPlanner.CurlingGaitFromSlipPlanner.SpeedDownFinished, style: Lamp-Lamp1-Yellow
    Lamp1 (933,436 27x29), variable: GVL.gaitPlanner.CurlingGaitFromSlipPlanner.MlegRollCFinished, style: Lamp-Lamp1-Yellow
    Lamp1 (933,463 27x29), variable: GVL.gaitPlanner.CurlingGaitFromSlipPlanner.AddHeightFinished, style: Lamp-Lamp1-Yellow
    Lamp1 (933,490 27x29), variable: GVL.gaitPlanner.CurlingGaitFromSlipPlanner.FlegRotBFinished, style: Lamp-Lamp1-Yellow
    Lamp1 (933,541 27x29), variable: GVL.gaitPlanner.CurlingGaitFromSlipPlanner.CurlingGaitFinished, style: Lamp-Lamp1-Yellow
    Lamp1 (933,31 27x29), variable: GVL.gaitPlanner.CurlingGaitFromSlipPlanner.ReadyFinished, style: Lamp-Lamp1-Yellow
    Label (700,220 107x30), "MlegRollB"
    Label (700,193 107x30), "OrientAdjust"
    Label (700,108 107x30), "BLegPosAdjust"
    Button (962,247 84x23), "Rep SR"
        toggle GVL.gaitPlanner.CurlingGaitFromSlipPlanner.RequireRepeateStoneRot
    Button (962,192 84x23), "Rep OA"
        toggle GVL.gaitPlanner.CurlingGaitFromSlipPlanner.RequireRepeateOrientAdjust
    Button (962,108 84x23), "Rep BLPA"
        toggle GVL.gaitPlanner.CurlingGaitFromSlipPlanner.RequireRepeateBLegPosAdjust
    Button (962,80 84x23), "Rep BPA"
        toggle GVL.gaitPlanner.CurlingGaitFromSlipPlanner.RequireRepeateBodyPosAdjust
    GroupBox (1055,10 236x586), "Trot control"
        Label (8,21 107x30), "Trgt Trot Vel"
        Label (8,54 107x30), "Trgt Side Vel"
        Label (8,87 107x30), "Trgt Turn Vel"
        Textfield (108,26 113x24), "%.3f", text variable: GVL.TrotWalk_trot_vel_desire
            OnMouseClick: write the text variable via Default
        Textfield (108,59 113x24), "%.3f", text variable: GVL.TrotWalk_side_vel_desire
            OnMouseClick: write the text variable via Default
        Textfield (108,92 113x24), "%.3f", text variable: GVL.TrotWalk_turn_rate_desire
            OnMouseClick: write the text variable via Default
        Label (8,120 107x30), "Cur Trot Vel (A)"
        Label (8,153 107x30), "Cur Side Vel (A)"
        Label (8,186 107x30), "Cur Turn Vel (A)"
        Textfield (108,125 113x24), "%.3f", text variable: GVL.gaitPlanner.TrotWalkPlanner.trot_vel[0]
        Textfield (108,158 113x24), "%.3f", text variable: GVL.gaitPlanner.TrotWalkPlanner.side_vel[0]
        Textfield (108,191 113x24), "%.3f", text variable: GVL.gaitPlanner.TrotWalkPlanner.turn_rate[0]
        Label (8,316 107x30), "Trot Step"
        Label (8,349 107x30), "Side Step"
        Label (8,379 107x30), "Turn Step"
        Textfield (108,321 113x24), "%.3f", text variable: GVL.TrotWalk_step[0]
            OnMouseClick: write the text variable via Default
        Textfield (108,354 113x24), "%.3f", text variable: GVL.TrotWalk_step[1]
            OnMouseClick: write the text variable via Default
        Textfield (108,385 113x24), "%.3f", text variable: GVL.TrotWalk_step[2]
            OnMouseClick: write the text variable via Default
        Button (11,557 66x23), "Req Move"
            toggle GVL.gaitPlanner.TrotWalkPlanner.require_move
        Button (83,557 66x23), "Req Stop"
            toggle GVL.gaitPlanner.TrotWalkPlanner.require_stop
        Button (155,557 74x23), "Quit"
            toggle GVL.gaitPlanner.TrotWalkPlanner.quit_flag
        Label (8,524 107x30), "In TrotWalk"
        Lamp1 (107,525 27x29), variable: GVL.gaitPlanner.TrotWalkPlanner.inTrot[0], style: Lamp-Lamp1-Yellow
        Label (8,219 107x30), "Cur Trot Vel (B)"
        Lamp1 (147,525 27x29), variable: GVL.gaitPlanner.TrotWalkPlanner.inTrot[1], style: Lamp-Lamp1-Yellow
        Lamp1 (193,525 27x29), variable: GVL.gaitPlanner.TrotWalkPlanner.isTrotWalk, style: Lamp-Lamp1-Green
        Label (7,411 107x30), "Period"
    Label (1063,31 107x30), "Trgt Trot Vel"
    Label (1063,64 107x30), "Trgt Side Vel"
    Label (1063,97 107x30), "Trgt Turn Vel"
    Textfield (1163,36 113x24), "%.3f", text variable: GVL.TrotWalk_trot_vel_desire
        OnMouseClick: write the text variable via Default, min -0.35, max 0.35
    Textfield (1163,69 113x24), "%.3f", text variable: GVL.TrotWalk_side_vel_desire
        OnMouseClick: write the text variable via Default, min -0.2, max 0.2
    Textfield (1163,102 113x24), "%.3f", text variable: GVL.TrotWalk_turn_rate_desire
        OnMouseClick: write the text variable via Default, min -0.2, max 0.2
    Label (1063,130 107x30), "Cur Trot Vel (A)"
    Label (1063,163 107x30), "Cur Side Vel (A)"
    Label (1063,196 107x30), "Cur Turn Vel (A)"
    Textfield (1163,135 113x24), "%.3f", text variable: GVL.gaitPlanner.TrotWalkPlanner.trot_vel[0]
    Textfield (1163,168 113x24), "%.3f", text variable: GVL.gaitPlanner.TrotWalkPlanner.side_vel[0]
    Textfield (1163,201 113x24), "%.3f", text variable: GVL.gaitPlanner.TrotWalkPlanner.turn_rate[0]
    Label (1063,326 107x30), "Trot Step"
    Label (1063,359 107x30), "Side Step"
    Label (1063,389 107x30), "Turn Step"
    Textfield (1163,331 113x24), "%.3f", text variable: GVL.TrotWalk_step[0]
        OnMouseClick: write the text variable via Default
    Textfield (1163,364 113x24), "%.3f", text variable: GVL.TrotWalk_step[1]
        OnMouseClick: write the text variable via Default
    Textfield (1163,395 113x24), "%.3f", text variable: GVL.TrotWalk_step[2]
        OnMouseClick: write the text variable via Default
    Button (1066,567 66x23), "Req Move"
        toggle GVL.gaitPlanner.TrotWalkPlanner.require_move
    Button (1138,567 66x23), "Req Stop"
        toggle GVL.gaitPlanner.TrotWalkPlanner.require_stop
    Button (1210,567 74x23), "Quit"
        toggle GVL.gaitPlanner.TrotWalkPlanner.quit_flag
    Label (1063,534 107x30), "In TrotWalk"
    Lamp1 (1162,535 27x29), variable: GVL.gaitPlanner.TrotWalkPlanner.inTrot[0], style: Lamp-Lamp1-Yellow
    Label (1063,229 107x30), "Cur Trot Vel (B)"
    Lamp1 (1202,535 27x29), variable: GVL.gaitPlanner.TrotWalkPlanner.inTrot[1], style: Lamp-Lamp1-Yellow
    Lamp1 (1248,535 27x29), variable: GVL.gaitPlanner.TrotWalkPlanner.isTrotWalk, style: Lamp-Lamp1-Green
    Label (1062,421 107x30), "Period"
    Label (1063,262 107x30), "Cur Side Vel (B)"
    Label (1063,295 107x30), "Cur Turn Vel (B)"
    Textfield (1163,234 113x24), "%.3f", text variable: GVL.gaitPlanner.TrotWalkPlanner.trot_vel[1]
    Textfield (1163,267 113x24), "%.3f", text variable: GVL.gaitPlanner.TrotWalkPlanner.side_vel[1]
    Textfield (1163,300 113x24), "%.3f", text variable: GVL.gaitPlanner.TrotWalkPlanner.turn_rate[1]
    Label (1062,454 107x30), "Duty"
    Label (1062,488 107x30), "Step height"
    Textfield (1162,426 113x24), "%.3f", text variable: GVL.period_desire
        OnMouseClick: write the text variable via Default
    Textfield (1162,459 113x24), "%.3f", text variable: GVL.duty_desire
        OnMouseClick: write the text variable via Default
    Textfield (1162,490 113x24), "%.3f", text variable: GVL.step_height_desire
        OnMouseClick: write the text variable via Default
    Lamp1 (442,287 27x29), variable: GVL.gaitPlanner.CurlingGaitPlanner2.IsOrientAdjust, style: Lamp-Lamp1-Green
    Button (473,287 84x23), "Req MRB"
        toggle GVL.gaitPlanner.CurlingGaitPlanner2.RequireMlegRollB
    Lamp1 (568,286 27x29), variable: GVL.gaitPlanner.CurlingGaitPlanner2.OrientAdjustFinished, style: Lamp-Lamp1-Yellow
    Lamp1 (811,222 27x29), variable: GVL.gaitPlanner.CurlingGaitFromSlipPlanner.IsMlegRollB, style: Lamp-Lamp1-Green
    Button (842,221 84x23), "Req SR"
        toggle GVL.gaitPlanner.CurlingGaitFromSlipPlanner.RequireStoneRot
    Lamp1 (933,221 27x29), variable: GVL.gaitPlanner.CurlingGaitFromSlipPlanner.MlegRollBFinished, style: Lamp-Lamp1-Yellow
    Lamp1 (811,195 27x29), variable: GVL.gaitPlanner.CurlingGaitFromSlipPlanner.IsOrientAdjust, style: Lamp-Lamp1-Green
    Button (842,194 84x23), "Req MRB"
        toggle GVL.gaitPlanner.CurlingGaitFromSlipPlanner.RequireMlegRollB
    Lamp1 (933,194 27x29), variable: GVL.gaitPlanner.CurlingGaitFromSlipPlanner.OrientAdjustFinished, style: Lamp-Lamp1-Yellow
    Lamp1 (442,235 27x29), variable: GVL.gaitPlanner.CurlingGaitPlanner2.IsSearchPedal, style: Lamp-Lamp1-Green
    Button (473,234 84x23), "Req AC"
        toggle GVL.gaitPlanner.CurlingGaitPlanner2.RequireArmControl
    Lamp1 (568,234 27x29), variable: GVL.gaitPlanner.CurlingGaitPlanner2.SearchPedalFinished, style: Lamp-Lamp1-Yellow
    Button (600,182 84x23), "Rep BPA"
        toggle GVL.gaitPlanner.CurlingGaitPlanner2.RequireRepeateBodyPosAdjust
    Label (338,181 107x30), "BodyPosAdjust"
    Lamp1 (442,183 27x29), variable: GVL.gaitPlanner.CurlingGaitPlanner2.IsBodyPosAdjust, style: Lamp-Lamp1-Green
    Button (473,183 84x23), "Req BLPA"
        toggle GVL.gaitPlanner.CurlingGaitPlanner2.RequireBLegPosAdjust
    Lamp1 (568,182 27x29), variable: GVL.gaitPlanner.CurlingGaitPlanner2.BodyPosAdjustFinished, style: Lamp-Lamp1-Yellow
    Label (700,81 107x30), "BodyPosAdjust"
    Lamp1 (811,110 27x29), variable: GVL.gaitPlanner.CurlingGaitFromSlipPlanner.IsBLegPosAdjust, style: Lamp-Lamp1-Green
    Button (842,109 84x23), "Req SP"
        toggle GVL.gaitPlanner.CurlingGaitFromSlipPlanner.RequireSearchPedal
    Lamp1 (933,109 27x29), variable: GVL.gaitPlanner.CurlingGaitFromSlipPlanner.OrientAdjustFinished, style: Lamp-Lamp1-Yellow
    Lamp1 (811,83 27x29), variable: GVL.gaitPlanner.CurlingGaitFromSlipPlanner.IsBodyPosAdjust, style: Lamp-Lamp1-Green
    Button (842,82 84x23), "Req BLPA"
        toggle GVL.gaitPlanner.CurlingGaitFromSlipPlanner.RequireBLegPosAdjust
    Lamp1 (933,82 27x29), variable: GVL.gaitPlanner.CurlingGaitFromSlipPlanner.BodyPosAdjustFinished, style: Lamp-Lamp1-Yellow
    Lamp1 (442,611 27x29), variable: GVL.gaitPlanner.CurlingGaitPlanner2.IsRecovery, style: Lamp-Lamp1-Green
    Button (473,609 84x23), "Req RHB"
        toggle GVL.gaitPlanner.CurlingGaitPlanner2.RequireReduceHeightB
    Lamp1 (568,610 27x29), variable: GVL.gaitPlanner.CurlingGaitPlanner2.RecoveryFinished, style: Lamp-Lamp1-Yellow
    Lamp1 (442,209 27x29), variable: GVL.gaitPlanner.CurlingGaitPlanner2.IsBLegPosAdjust, style: Lamp-Lamp1-Green
    Button (473,209 84x23), "Req SP"
        toggle GVL.gaitPlanner.CurlingGaitPlanner2.RequireSearchPedal
    Lamp1 (568,208 27x29), variable: GVL.gaitPlanner.CurlingGaitPlanner2.BLegPosAdjustFinished, style: Lamp-Lamp1-Yellow
    Lamp1 (442,261 27x29), variable: GVL.gaitPlanner.CurlingGaitPlanner2.IsArmControl, style: Lamp-Lamp1-Green
    Button (473,260 84x23), "Req OA"
        toggle GVL.gaitPlanner.CurlingGaitPlanner2.RequireOrientAdjust
    Lamp1 (568,260 27x29), variable: GVL.gaitPlanner.CurlingGaitPlanner2.ArmControlFinished, style: Lamp-Lamp1-Yellow
    Label (329,840 116x30), "视觉运动(度)"
    Lamp1 (442,504 27x29), variable: GVL.gaitPlanner.CurlingGaitPlanner2.IsBLegRecovery, style: Lamp-Lamp1-Green
    Button (473,501 84x23), "Req MRC"
        toggle GVL.gaitPlanner.CurlingGaitPlanner2.RequireMlegRollC
    Lamp1 (568,503 27x29), variable: GVL.gaitPlanner.CurlingGaitPlanner2.BLegRecoveryFinished, style: Lamp-Lamp1-Yellow
    Button (962,136 84x23), "Rep SP"
        toggle GVL.gaitPlanner.CurlingGaitPlanner2.RequireRepeateSearchPedal
    Lamp1 (811,137 27x29), variable: GVL.gaitPlanner.CurlingGaitFromSlipPlanner.IsSearchPedal, style: Lamp-Lamp1-Green
    Button (842,136 84x23), "Req AC"
        toggle GVL.gaitPlanner.CurlingGaitFromSlipPlanner.RequireArmControl
    Lamp1 (933,136 27x29), variable: GVL.gaitPlanner.CurlingGaitFromSlipPlanner.SearchPedalFinished, style: Lamp-Lamp1-Yellow
    Button (962,165 84x23), "Rep AC"
        toggle GVL.gaitPlanner.CurlingGaitPlanner2.RequireRepeateArmControl
    Lamp1 (811,166 27x29), variable: GVL.gaitPlanner.CurlingGaitFromSlipPlanner.IsArmControl, style: Lamp-Lamp1-Green
    Button (842,165 84x23), "Req OA"
        toggle GVL.gaitPlanner.CurlingGaitFromSlipPlanner.RequireOrientAdjust
    Lamp1 (933,165 27x29), variable: GVL.gaitPlanner.CurlingGaitFromSlipPlanner.ArmControlFinished, style: Lamp-Lamp1-Yellow
    Lamp1 (811,412 27x29), variable: GVL.gaitPlanner.CurlingGaitFromSlipPlanner.IsBLegRecovery, style: Lamp-Lamp1-Green
    Button (842,409 84x23), "Req MRC"
        toggle GVL.gaitPlanner.CurlingGaitFromSlipPlanner.RequireMlegRollC
    Lamp1 (933,411 27x29), variable: GVL.gaitPlanner.CurlingGaitFromSlipPlanner.BLegRecoveryFinished, style: Lamp-Lamp1-Yellow
    Lamp1 (811,516 27x29), variable: GVL.gaitPlanner.CurlingGaitFromSlipPlanner.IsRecovery, style: Lamp-Lamp1-Green
    Button (842,514 84x23), "Req CF"
        toggle GVL.gaitPlanner.CurlingGaitFromSlipPlanner.quit_flag
    Lamp1 (933,515 27x29), variable: GVL.gaitPlanner.CurlingGaitFromSlipPlanner.RecoveryFinished, style: Lamp-Lamp1-Yellow
    GroupBox (941,596 168x277), "斜坡行走"
        Textfield (87,69 70x30), "%.2f", text variable: GVL.gaitPlanner.WalkSlopePlanner.cmdL
            OnMouseClick: write the text variable via Default
        Textfield (87,174 70x30), "%.2f", text variable: GVL.gaitPlanner.WalkSlopePlanner.period
            OnMouseClick: write the text variable via Default
        Textfield (87,209 70x30), "%.2f", text variable: GVL.gaitPlanner.WalkSlopePlanner.cmdH
            OnMouseClick: write the text variable via Default
        Label (5,138 80x30), "转弯角度(度)"
        Textfield (87,139 70x30), "%.2f", text variable: GVL.gaitPlanner.WalkSlopePlanner.cmdYaw
            OnMouseClick: write the text variable via Default
        Button (17,26 129x30), "停止"
            toggle GVL.gaitPlanner.WalkSlopePlanner.isLastStep
        Textfield (87,104 70x30), "%.2f", text variable: GVL.gaitPlanner.WalkSlopePlanner.cmdLa
            OnMouseClick: write the text variable via Default
        Label (1,68 91x30), "前进步长"
        Textfield (87,243 70x30), "%d", text variable: GVL.gaitPlanner.WalkSlopePlanner.swingDir
            OnMouseClick: write the text variable via Default
        Label (0,241 90x30), "摆动方向"
    Textfield (1028,665 70x30), "%.2f", text variable: GVL.gaitPlanner.WalkSlopePlanner.cmdL
        OnMouseClick: write the text variable via Default
    Textfield (1028,770 70x30), "%.2f", text variable: GVL.gaitPlanner.WalkSlopePlanner.period
        OnMouseClick: write the text variable via Default
    Textfield (1028,805 70x30), "%.2f", text variable: GVL.gaitPlanner.WalkSlopePlanner.cmdH
        OnMouseClick: write the text variable via Default
    Label (946,734 80x30), "转弯角度(度)"
    Textfield (1028,735 70x30), "%.2f", text variable: GVL.gaitPlanner.WalkSlopePlanner.cmdYaw
        OnMouseClick: write the text variable via Default
    Button (958,622 129x30), "停止"
        toggle GVL.gaitPlanner.WalkSlopePlanner.isLastStep
    Textfield (1028,700 70x30), "%.2f", text variable: GVL.gaitPlanner.WalkSlopePlanner.cmdLa
        OnMouseClick: write the text variable via Default
    Label (942,664 91x30), "前进步长"
    Textfield (1028,839 70x30), "%d", text variable: GVL.gaitPlanner.WalkSlopePlanner.swingDir
        OnMouseClick: write the text variable via Default
    Label (941,837 90x30), "摆动方向"
    Label (946,772 80x30), "周期"
    Label (941,803 90x30), "步高"
    Label (940,698 92x30), "侧移步长"
    Textfield (1135,604 70x30), "%.2f", text variable: GVL.gaitPlanner.WalkSlopePlanner.kp
        OnMouseClick: write the text variable via Default
    Textfield (1133,644 70x30), "%.2f", text variable: GVL.gaitPlanner.WalkSlopePlanner.ki
        OnMouseClick: write the text variable via Default
    Textfield (1135,681 70x30), "%.2f", text variable: GVL.gaitPlanner.WalkSlopePlanner.kd
        OnMouseClick: write the text variable via Default
    Textfield (1218,605 70x30), "%.2f", text variable: GVL.gaitPlanner.WalkSlopePlanner.tipFce[0].data[2]
        OnMouseClick: write the text variable via Default
    Textfield (1216,645 70x30), "%.2f", text variable: GVL.gaitPlanner.WalkSlopePlanner.tipFce[1].data[2]
        OnMouseClick: write the text variable via Default
    Textfield (1218,682 70x30), "%.2f", text variable: GVL.gaitPlanner.WalkSlopePlanner.tipFce[2].data[2]
        OnMouseClick: write the text variable via Default
    Textfield (1219,719 70x30), "%.2f", text variable: GVL.gaitPlanner.WalkSlopePlanner.tipFce[3].data[2]
        OnMouseClick: write the text variable via Default
    Textfield (1217,759 70x30), "%.2f", text variable: GVL.gaitPlanner.WalkSlopePlanner.tipFce[4].data[2]
        OnMouseClick: write the text variable via Default
    Textfield (1219,796 70x30), "%.2f", text variable: GVL.gaitPlanner.WalkSlopePlanner.tipFce[5].data[2]
        OnMouseClick: write the text variable via Default
    Textfield (1135,727 70x30), "%.2f", text variable: GVL.gaitPlanner.WalkSlopePlanner.kRatio
        OnMouseClick: write the text variable via Default
    Lamp1 (443,636 27x29), variable: GVL.gaitPlanner.CurlingGaitPlanner2.IsReduceHeightB, style: Lamp-Lamp1-Green
    Button (474,634 84x23), "Req CF"
        toggle GVL.gaitPlanner.CurlingGaitPlanner2.quit_flag
    Lamp1 (569,635 27x29), variable: GVL.gaitPlanner.CurlingGaitPlanner2.ReduceHeightBFinished, style: Lamp-Lamp1-Yellow
    Lamp1 (443,53 27x29), variable: GVL.gaitPlanner.CurlingGaitPlanner2.IsReady, style: Lamp-Lamp1-Green
    Button (474,53 84x23), "Req BC"
        toggle GVL.gaitPlanner.CurlingGaitPlanner2.RequireBlegCenter
    Lamp1 (569,53 27x29), variable: GVL.gaitPlanner.CurlingGaitPlanner2.ReadyFinished, style: Lamp-Lamp1-Yellow
    Lamp1 (443,53 27x29), variable: GVL.gaitPlanner.CurlingGaitPlanner2.IsAddHeightFromWalk, style: Lamp-Lamp1-Green
    Button (474,53 84x23), "Req BC"
        toggle GVL.gaitPlanner.CurlingGaitPlanner2.RequireBlegCenter
    Lamp1 (569,53 27x29), variable: GVL.gaitPlanner.CurlingGaitPlanner2.AddHeightFromWalkFinished, style: Lamp-Lamp1-Yellow
END_VISUALIZATION

(* stored: Version 1.1.0.1, ProductVersion 3.1.4024.2
   Visu RobotUI: Id {3f107c53-f61f-43ad-9977-e0c439fb3f04} *)
